// TIA Portal V20 export
TYPE "TypeBaluffBUS007xRd"
   STRUCT
      Measure : Int;   // Actual measured value 300...3500 1/10mm (-1= Read error)
      Scale : SInt;   // Scale -1 = 1/10mm
      SCC1 : Bool;   // Signal output 1 (1= Occ)
      res1 : Bool;
      res2 : Bool;
      res3 : Bool;
      res4 : Bool;
      res5 : Bool;
      res6 : Bool;
      res7 : Bool;
   END_STRUCT;
END_TYPE
